KUKA KRL program: saco_20_m2.src, saco_20_m2.dat

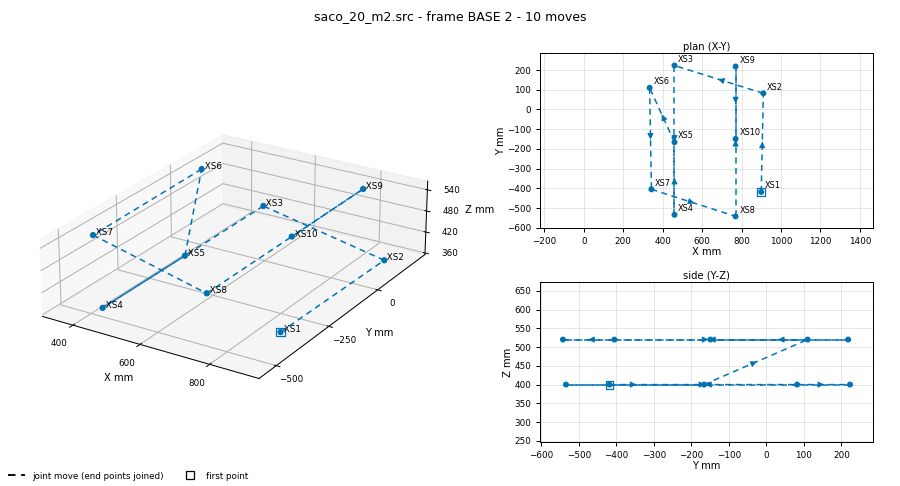
[picture p0: tool path of saco_20_m2.src in frame BASE 2, 10 of 19 moves have a stored position in this frame; points joined in program order, loops and branches not executed]
--- saco_20_m2.src ---
&ACCESS RVO1
&REL 89
&PARAM DISKPATH = KRC:\R1\Program\SACO_20
&PARAM TEMPLATE = C:\KRC\Roboter\Template\vorgabe
&PARAM EDITMASK = *
DEF saco_20_M2( )
;Fold DECLARACION VARIABLES
DECL E6POS POS_A
DECL E6POS POS_B
DECL E6POS POS_C
DECL REAL INC_Z
DECL INT PLANTA
DECL INT SACOS_A_PALETIZAR
DECL E6POS PUNTO[10]
DECL INT n
EXT COGE_20 ()
;Endfold
;FOLD INI;%{PE}
  ;FOLD BASISTECH INI
    GLOBAL INTERRUPT DECL 3 WHEN $STOPMESS==TRUE DO IR_STOPM ( )
    INTERRUPT ON 3
    BAS (#INITMOV,0 )
  ;ENDFOLD (BASISTECH INI)
;FOLD SPOTTECH INI
USERSPOT(#INIT)
;ENDFOLD (SPOTTECH INI)
;FOLD GRIPPERTECH INI
USER_GRP(0,DUMMY,DUMMY,GDEFAULT)
;ENDFOLD (GRIPPERTECH INI)
  ;FOLD USER INI
    ;Make your modifications here

  ;ENDFOLD (USER INI)
;ENDFOLD (INI)
; === PROGRAMA PALETIZADO 50 SACOS ARYSTA 20 KG MOSAICO 5-5 ==
;Fold VARIABLES
INC_Z=0
PLANTA = 1
N_SACO=0
SACOS_A_PALETIZAR=50
n=1
PUNTO[1]=XS1
PUNTO[2]=XS2
PUNTO[3]=XS3
PUNTO[4]=XS4
PUNTO[5]=XS5
PUNTO[6]=XS6
PUNTO[7]=XS7
PUNTO[8]=XS8
PUNTO[9]=XS9
PUNTO[10]=XS10
;Endfold
;FOLD PTP HOME  Vel= 100 % DEFAULT;%{PE}%MKUKATPBASIS,%CMOVE,%VPTP,%P 1:PTP, 2:HOME, 3:, 5:100, 7:DEFAULT
$BWDSTART = FALSE
PDAT_ACT=PDEFAULT
FDAT_ACT=FHOME
BAS (#PTP_PARAMS,100 )
$H_POS=XHOME
PTP  XHOME
;ENDFOLD
;Fold Compruebo Palet
WAIT FOR PALET_LIBRE OR SALIR_PROGRAMA_ACTUAL
IF SALIR_PROGRAMA_ACTUAL == TRUE THEN
   PULSE ( OK_LEIDO_SALIR_PROGRAMA, true, 0.5 )
   WAIT SEC 1
   GOTO SALIRPROG
ENDIF
;Endfold
BOMBA =TRUE
;=== BUCLE PRINCIPAL ==
FOR PLANTA=1 TO 12 ;Bucle de plantas
FOR n=1 TO 10 ;Bucle de sacos
SACO:

;Fold WAIT FOR REPITE_SACO: Espero repetir saco si ha caido
IF (ERROR_SACO_CAIDO == TRUE ) THEN
   WAIT FOR REPITE_SACO OR SALIR_PROGRAMA_ACTUAL
   ERROR_SACO_CAIDO = FALSE
ENDIF
;Endfold

;Fold DEFINICION PUNTOS AUXILIARES
POS_A =PUNTO[n]
POS_B =PUNTO[n]
POS_C =PUNTO[n]

POS_A.Z=POS_A.Z+INC_Z+400
POS_B.Z=POS_B.Z+INC_Z+250
POS_C.Z=POS_C.Z+INC_Z+0

;Endfold

COGE_20 () ;Llamo programa coger
;Fold CONDICION DE SALIDA DE PROGRAMA PLC
IF SALIR == TRUE THEN
   GOTO SALIRPROG
ENDIF
;Endfold

BAS(#BASE,2) ;Cambio de base
$APO.CPTP = 70

;Fold Velocidad SACO 20 Kg
FOR ax_num=1 TO 6
$VEL_AXIS[ax_num]=vptpSACO20
$ACC_AXIS[ax_num]=vaccSACO20
ENDFOR
$VEL.CP=vlinSACO20
;Endfold

;Fold Bajo velocidad Saco 4
Continue
IF (n==4) THEN
FOR ax_num=1 TO 6
$VEL_AXIS[ax_num]=20
$ACC_AXIS[ax_num]=20
ENDFOR
$VEL.CP=0.5
ENDIF
;Endfold

;Fold Bajo velocidad Saco 5
Continue
IF (n==5) THEN
FOR ax_num=1 TO 6
$VEL_AXIS[ax_num]=20
$ACC_AXIS[ax_num]=20
ENDFOR
$VEL.CP=0.5
ENDIF
;Endfold

PTP POS_A C_PTP

PTP POS_B C_PTP

;Fold Velocidad Lenta
FOR ax_num=1 TO 6
$VEL_AXIS[ax_num]=vptpL
$ACC_AXIS[ax_num]=vaccL
ENDFOR
$VEL.CP=vlinL
;Endfold

LIN POS_C

;Fold Compruebo caida de saco
IF (VACOESTATO == FALSE) THEN ;Condicion de saco perdido
   ERROR_SACO_CAIDO = TRUE
   FOR ax_num=1 TO 6
   $VEL_AXIS[ax_num]=vptpR
   $ACC_AXIS[ax_num]=vaccR
   ENDFOR
   $VEL.CP=vlinR
   LIN POS_A
   ;FOLD PTP HOME  Vel= 100 % DEFAULT;%{PE}%MKUKATPBASIS,%CMOVE,%VPTP,%P 1:PTP, 2:HOME, 3:, 5:100, 7:DEFAULT
$BWDSTART = FALSE
PDAT_ACT=PDEFAULT
FDAT_ACT=FHOME
BAS (#PTP_PARAMS,100 )
$H_POS=XHOME
PTP  XHOME
;ENDFOLD
   GOTO SACO
ENDIF
;Endfold

WAIT SEC 0.2
VACIO=FALSE  ;Abro vacio
WAIT FOR NOT VACOESTATO OR VOLVER_COGER ;Espero Vacoestato

;Fold Velocidad Rapida
Continue
FOR ax_num=1 TO 6
$VEL_AXIS[ax_num]=vptpR
$ACC_AXIS[ax_num]=vaccR
ENDFOR
$VEL.CP=vlinR
;Endfold

LIN POS_A C_DIS

;FOLD PTP HOME CONT Vel=ptpM % DEFAULT;%{PE}%R 8.2.24,%MKUKATPBASIS,%CMOVE,%VPTP,%P 1:PTP, 2:HOME, 3:C_DIS, 5:50, 7:DEFAULT
$BWDSTART=FALSE
PDAT_ACT=PDEFAULT
FDAT_ACT=FHOME
BAS(#PTP_PARAMS,vptpM)
$H_POS=XHOME
$APO.CPTP = 70
PTP XHOME C_PTP
;ENDFOLD

;Fold Incremento Saco
N_SACO=N_SACO+1
IF (N_SACO >= SACOS_A_PALETIZAR) THEN
   GOTO FINAL
ENDIF
;Endfold

ENDFOR

;Fold Incremento Planta
PLANTA = PLANTA + 1

IF PLANTA <=2 THEN
INC_Z=INC_Z+190.0 ;Incremento cota superior
ENDIF

IF PLANTA >3 THEN
INC_Z=INC_Z+180.0 ;Incremento cota superior
ENDIF

;Endfold

ENDFOR


GOTO FINAL
;Fold PUNTOS COGIDA SOLO PARA MODIFICAR TOUCHAP
;FOLD PTP S1 Vel=50 % PDAT1 Tool[1]:VENTOSA_SACOS Base[2]:PALETS;%{PE}%R 8.2.24,%MKUKATPBASIS,%CMOVE,%VPTP,%P 1:PTP, 2:S1, 3:, 5:100, 7:PDAT1
$BWDSTART=FALSE
PDAT_ACT=PPDAT1
FDAT_ACT=FS1
BAS(#PTP_PARAMS,50)
PTP XS1
;ENDFOLD
;FOLD PTP S2 Vel=50 % PDAT2 Tool[1]:VENTOSA_SACOS Base[2]:PALETS;%{PE}%R 8.2.24,%MKUKATPBASIS,%CMOVE,%VPTP,%P 1:PTP, 2:S2, 3:, 5:100, 7:PDAT2
$BWDSTART=FALSE
PDAT_ACT=PPDAT2
FDAT_ACT=FS2
BAS(#PTP_PARAMS,50)
PTP XS2
;ENDFOLD
;FOLD PTP S3 Vel=50 % PDAT3 Tool[1]:VENTOSA_SACOS Base[2]:PALETS;%{PE}%R 8.2.24,%MKUKATPBASIS,%CMOVE,%VPTP,%P 1:PTP, 2:S3, 3:, 5:100, 7:PDAT3
$BWDSTART=FALSE
PDAT_ACT=PPDAT3
FDAT_ACT=FS3
BAS(#PTP_PARAMS,50)
PTP XS3
;ENDFOLD
;FOLD PTP S4 Vel=50 % PDAT4 Tool[1]:VENTOSA_SACOS Base[2]:PALETS;%{PE}%R 8.2.24,%MKUKATPBASIS,%CMOVE,%VPTP,%P 1:PTP, 2:S4, 3:, 5:100, 7:PDAT4
$BWDSTART=FALSE
PDAT_ACT=PPDAT4
FDAT_ACT=FS4
BAS(#PTP_PARAMS,50)
PTP XS4
;ENDFOLD
;FOLD PTP S5 Vel=50 % PDAT5 Tool[1]:VENTOSA_SACOS Base[2]:PALETS;%{PE}%R 8.2.24,%MKUKATPBASIS,%CMOVE,%VPTP,%P 1:PTP, 2:S5, 3:, 5:100, 7:PDAT5
$BWDSTART=FALSE
PDAT_ACT=PPDAT5
FDAT_ACT=FS5
BAS(#PTP_PARAMS,50)
PTP XS5
;ENDFOLD
;FOLD PTP S6 Vel=50 % PDAT6 Tool[1]:VENTOSA_SACOS Base[2]:PALETS;%{PE}%R 8.2.24,%MKUKATPBASIS,%CMOVE,%VPTP,%P 1:PTP, 2:S6, 3:, 5:100, 7:PDAT6
$BWDSTART=FALSE
PDAT_ACT=PPDAT6
FDAT_ACT=FS6
BAS(#PTP_PARAMS,50)
PTP XS6
;ENDFOLD
;FOLD PTP S7 Vel=50 % PDAT7 Tool[1]:VENTOSA_SACOS Base[2]:PALETS;%{PE}%R 8.2.24,%MKUKATPBASIS,%CMOVE,%VPTP,%P 1:PTP, 2:S7, 3:, 5:100, 7:PDAT7
$BWDSTART=FALSE
PDAT_ACT=PPDAT7
FDAT_ACT=FS7
BAS(#PTP_PARAMS,50)
PTP XS7
;ENDFOLD
;FOLD PTP S8 Vel=50 % PDAT8 Tool[1]:VENTOSA_SACOS Base[2]:PALETS;%{PE}%R 8.2.24,%MKUKATPBASIS,%CMOVE,%VPTP,%P 1:PTP, 2:S8, 3:, 5:100, 7:PDAT8
$BWDSTART=FALSE
PDAT_ACT=PPDAT8
FDAT_ACT=FS8
BAS(#PTP_PARAMS,50)
PTP XS8
;ENDFOLD
;FOLD PTP S9 Vel=50 % PDAT9 Tool[1]:VENTOSA_SACOS Base[2]:PALETS;%{PE}%R 8.2.24,%MKUKATPBASIS,%CMOVE,%VPTP,%P 1:PTP, 2:S9, 3:, 5:100, 7:PDAT9
$BWDSTART=FALSE
PDAT_ACT=PPDAT9
FDAT_ACT=FS9
BAS(#PTP_PARAMS,50)
PTP XS9
;ENDFOLD
;FOLD PTP S10 Vel=50 % PDAT10 Tool[1]:VENTOSA_SACOS Base[2]:PALETS;%{PE}%R 8.2.24,%MKUKATPBASIS,%CMOVE,%VPTP,%P 1:PTP, 2:S10, 3:, 5:100, 7:PDAT10
$BWDSTART=FALSE
PDAT_ACT=PPDAT10
FDAT_ACT=FS10
BAS(#PTP_PARAMS,50)
PTP XS10
;ENDFOLD

;Endfold

FINAL:

PULSE ( PALET_COMPLETO, TRUE, 0.5 )
WAIT SEC 1

SALIRPROG:

N_SACO=0
SALIR=FALSE
BOMBA=FALSE

;FOLD PTP HOME CONT Vel=ptpM % DEFAULT;%{PE}%R 8.2.24,%MKUKATPBASIS,%CMOVE,%VPTP,%P 1:PTP, 2:HOME, 3:C_DIS, 5:50, 7:DEFAULT
$BWDSTART=FALSE
PDAT_ACT=PDEFAULT
FDAT_ACT=FHOME
BAS(#PTP_PARAMS,vptpM)
$H_POS=XHOME
$APO.CPTP = 70
PTP XHOME C_PTP
;ENDFOLD

END

--- saco_20_m2.dat ---
&ACCESS RVO1
&REL 89
&PARAM DISKPATH = KRC:\R1\Program\SACO_20
&PARAM TEMPLATE = C:\KRC\Roboter\Template\vorgabe
&PARAM EDITMASK = *
DEFDAT  saco_20_m2
;FOLD EXTERNAL DECLARATIONS;%{PE}%MKUKATPBASIS,%CEXT,%VCOMMON,%P
;FOLD GRIPPERTECH EXT
EXT  H50 (INT  :IN,INT  :IN,INT  :IN,GRP_TYP  :IN )
;ENDFOLD (GRIPPERTECH EXT)
;FOLD SPOTTECH EXT
EXT  USERSPOT (S_COMMAND  :IN,SPOT_TYPE  :IN )
;ENDFOLD (SPOTTECH EXT)
;FOLD BASISTECH EXT;%{PE}%MKUKATPBASIS,%CEXT,%VEXT,%P
EXT  BAS (BAS_COMMAND  :IN,REAL  :IN )
DECL INT SUCCESS
;ENDFOLD (BASISTECH EXT)
;FOLD USER EXT;%{E}%MKUKATPUSER,%CEXT,%VEXT,%P
;Make your modifications here

;ENDFOLD (USER EXT)
;ENDFOLD (EXTERNAL DECLARATIONS)
DECL BASIS_SUGG_T LAST_BASIS={POINT1[] "BOX                     ",POINT2[] "BOX                     ",CP_PARAMS[] "CPDAT0                  ",PTP_PARAMS[] "PDAT28                  ",CONT[] "C_DIS                   ",CP_VEL[] "2.0                     ",PTP_VEL[] "50                      ",SYNC_PARAMS[] "SYNCDAT                 ",SPL_NAME[] "S0                      "}

DECL E6POS XS1={X 900,Y -417.978485,Z 400,A 177.897003,B -0.195673898,C -179.634796,S 2,T 11,E1 0.0,E2 0.0,E3 0.0,E4 0.0,E5 0.0,E6 0.0}
DECL FDAT FS1={TOOL_NO 1,BASE_NO 2,IPO_FRAME #BASE,POINT2[] " ",TQ_STATE FALSE}
DECL PDAT PPDAT1={VEL 100.0,ACC 100.0,APO_DIST 100.0,APO_MODE #CDIS,GEAR_JERK 50.0}
DECL E6POS XS2={X 910.78363,Y 81.9997635,Z 400.001099,A -3.19985795,B 0.187563106,C 179.6306,S 2,T 35,E1 0.0,E2 0.0,E3 0.0,E4 0.0,E5 0.0,E6 0.0}
DECL FDAT FS2={TOOL_NO 1,BASE_NO 2,IPO_FRAME #BASE,POINT2[] " ",TQ_STATE FALSE}
DECL PDAT PPDAT2={VEL 100.0,ACC 100.0,APO_DIST 100.0,APO_MODE #CDIS,GEAR_JERK 50.0}

DECL E6POS XS3={X 460.0,Y 223.0,Z 400.0,A 86.5,B 0.370000005,C -179.809998,S 2,T 43,E1 0.0,E2 0.0,E3 0.0,E4 0.0,E5 0.0,E6 0.0}
DECL FDAT FS3={TOOL_NO 1,BASE_NO 2,IPO_FRAME #BASE,POINT2[] " ",TQ_STATE FALSE}
DECL PDAT PPDAT3={VEL 100.0,ACC 100.0,APO_DIST 100.0,APO_MODE #CDIS,GEAR_JERK 50.0}
DECL E6POS XS4={X 460.0,Y -534.0,Z 400.0,A 86.5,B 0.370000005,C -179.809998,S 2,T 43,E1 0.0,E2 0.0,E3 0.0,E4 0.0,E5 0.0,E6 0.0}
DECL FDAT FS4={TOOL_NO 1,BASE_NO 2,IPO_FRAME #BASE,POINT2[] " ",TQ_STATE FALSE}
DECL PDAT PPDAT4={VEL 100.0,ACC 100.0,APO_DIST 100.0,APO_MODE #CDIS,GEAR_JERK 50.0}
DECL E6POS XS5={X 460.0,Y -166.0,Z 400.0,A 86.5,B 0.370000005,C -179.809998,S 2,T 43,E1 0.0,E2 0.0,E3 0.0,E4 0.0,E5 0.0,E6 0.0}
DECL FDAT FS5={TOOL_NO 1,BASE_NO 2,IPO_FRAME #BASE,POINT2[] " ",TQ_STATE FALSE}
DECL PDAT PPDAT5={VEL 100.0,ACC 100.0,APO_DIST 100.0,APO_MODE #CDIS,GEAR_JERK 50.0}

DECL E6POS XS6={X 334.0,Y 110.0,Z 520.0,A -3.53999996,B 0.180000007,C 179.619995,S 2,T 35,E1 0.0,E2 0.0,E3 0.0,E4 0.0,E5 0.0,E6 0.0}
DECL FDAT FS6={TOOL_NO 1,BASE_NO 2,IPO_FRAME #BASE,POINT2[] " ",TQ_STATE FALSE}
DECL PDAT PPDAT6={VEL 100.0,ACC 100.0,APO_DIST 100.0,APO_MODE #CDIS,GEAR_JERK 50.0}
DECL E6POS XS7={X 343.0,Y -405.0,Z 520.0,A 176.460007,B -0.180000007,C -179.619995,S 2,T 11,E1 0.0,E2 0.0,E3 0.0,E4 0.0,E5 0.0,E6 0.0}
DECL FDAT FS7={TOOL_NO 1,BASE_NO 2,IPO_FRAME #BASE,POINT2[] " ",TQ_STATE FALSE}
DECL PDAT PPDAT7={VEL 100.0,ACC 100.0,APO_DIST 100.0,APO_MODE #CDIS,GEAR_JERK 50.0}

DECL E6POS XS8={X 770.0,Y -542.0,Z 520.0,A -95.3399963,B -0.370000005,C 179.820007,S 2,T 3,E1 0.0,E2 0.0,E3 0.0,E4 0.0,E5 0.0,E6 0.0}
DECL FDAT FS8={TOOL_NO 1,BASE_NO 2,IPO_FRAME #BASE,POINT2[] " ",TQ_STATE FALSE}
DECL PDAT PPDAT8={VEL 100.0,ACC 100.0,APO_DIST 100.0,APO_MODE #CDIS,GEAR_JERK 50.0}
DECL E6POS XS9={X 770.0,Y 218.0,Z 520.0,A -94.5899963,B -0.370000005,C 179.820007,S 2,T 3,E1 0.0,E2 0.0,E3 0.0,E4 0.0,E5 0.0,E6 0.0}
DECL FDAT FS9={TOOL_NO 1,BASE_NO 2,IPO_FRAME #BASE,POINT2[] " ",TQ_STATE FALSE}
DECL PDAT PPDAT9={VEL 100.0,ACC 100.0,APO_DIST 100.0,APO_MODE #CDIS,GEAR_JERK 50.0}
DECL E6POS XS10={X 770.0,Y -149.0,Z 520.0,A -93.75,B -0.370000005,C 179.809998,S 2,T 3,E1 0.0,E2 0.0,E3 0.0,E4 0.0,E5 0.0,E6 0.0}
DECL FDAT FS10={TOOL_NO 1,BASE_NO 2,IPO_FRAME #BASE,POINT2[] " ",TQ_STATE FALSE}
DECL PDAT PPDAT10={VEL 100.0,ACC 100.0,APO_DIST 100.0,APO_MODE #CDIS,GEAR_JERK 50.0}

ENDDAT
